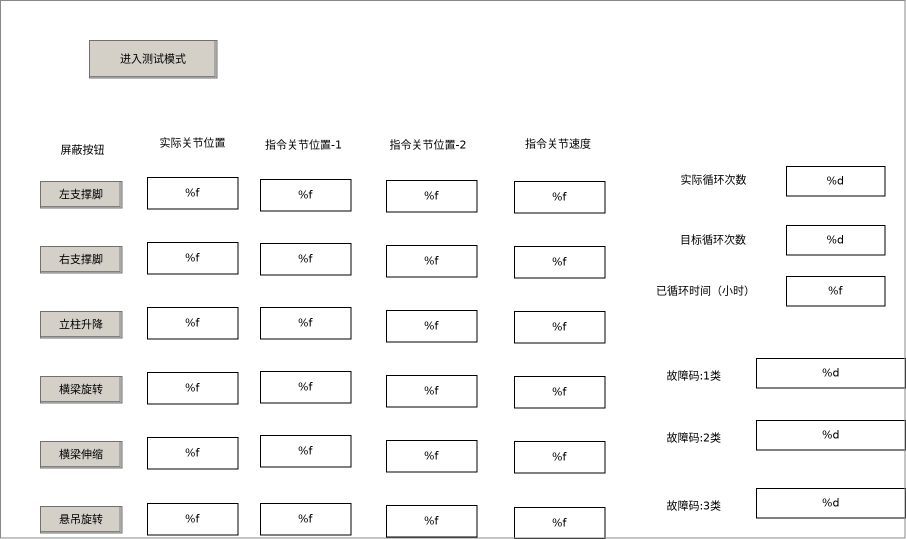
VISUALIZATION cartCycleTest  // 906x539
    Label (142,128 101x30), "实际关节位置"
    Rectangle (147,177 91x32), "%f", text variable: g_systemInfo.m_cartJntInfo[1].m_curJntPos
    Label (254,130 99x30), "指令关节位置-1"
    Button (89,40 128x38), "进入测试模式", colour toggle: g_cycleTest.m_carEnterCycleTest
        toggle g_cycleTest.m_carEnterCycleTest
    Rectangle (147,242 91x32), "%f", text variable: g_systemInfo.m_cartJntInfo[2].m_curJntPos
    Rectangle (260,179 91x32), "%f", text variable: g_cycleTest.m_targetJntPosCar[1][1]
        OnMouseClick: write the text variable via Default
    Rectangle (260,243 91x32), "%f", text variable: g_cycleTest.m_targetJntPosCar[1][2]
        OnMouseClick: write the text variable via Default
    Label (370,130 116x30), "指令关节位置-2"
    Rectangle (386,180 91x32), "%f", text variable: g_cycleTest.m_targetJntPosCar[2][1]
        OnMouseClick: write the text variable via Default
    Rectangle (386,245 91x32), "%f", text variable: g_cycleTest.m_targetJntPosCar[2][2]
        OnMouseClick: write the text variable via Default
    Rectangle (147,307 91x32), "%f", text variable: g_systemInfo.m_cartJntInfo[5].m_curJntPos
    Rectangle (147,372 91x32), "%f", text variable: g_systemInfo.m_cartJntInfo[6].m_curJntPos
    Rectangle (147,437 91x32), "%f", text variable: g_systemInfo.m_cartJntInfo[7].m_curJntPos
    Rectangle (147,503 91x32), "%f", text variable: g_systemInfo.m_cartJntInfo[8].m_curJntPos
    Rectangle (260,307 91x32), "%f", text variable: g_cycleTest.m_targetJntPosCar[1][5]
        OnMouseClick: write the text variable via Default
    Rectangle (260,371 91x32), "%f", text variable: g_cycleTest.m_targetJntPosCar[1][6]
        OnMouseClick: write the text variable via Default
    Rectangle (260,435 91x32), "%f", text variable: g_cycleTest.m_targetJntPosCar[1][7]
        OnMouseClick: write the text variable via Default
    Rectangle (260,503 91x32), "%f", text variable: g_cycleTest.m_targetJntPosCar[1][8]
        OnMouseClick: write the text variable via Default
    Rectangle (386,310 91x32), "%f", text variable: g_cycleTest.m_targetJntPosCar[2][5]
        OnMouseClick: write the text variable via Default
    Rectangle (386,375 91x32), "%f", text variable: g_cycleTest.m_targetJntPosCar[2][6]
        OnMouseClick: write the text variable via Default
    Rectangle (386,440 91x32), "%f", text variable: g_cycleTest.m_targetJntPosCar[2][7]
        OnMouseClick: write the text variable via Default
    Rectangle (386,505 91x32), "%f", text variable: g_cycleTest.m_targetJntPosCar[2][8]
        OnMouseClick: write the text variable via Default
    Label (507,130 102x28), "指令关节速度"
    Rectangle (514,181 91x32), "%f", text variable: g_cycleTest.m_targetJntVelCar[1]
        OnMouseClick: write the text variable via Default
    Rectangle (514,246 91x32), "%f", text variable: g_cycleTest.m_targetJntVelCar[2]
        OnMouseClick: write the text variable via Default
    Rectangle (514,311 91x32), "%f", text variable: g_cycleTest.m_targetJntVelCar[5]
        OnMouseClick: write the text variable via Default
    Rectangle (514,376 91x32), "%f", text variable: g_cycleTest.m_targetJntVelCar[6]
        OnMouseClick: write the text variable via Default
    Rectangle (514,441 91x32), "%f", text variable: g_cycleTest.m_targetJntVelCar[7]
        OnMouseClick: write the text variable via Default
    Rectangle (514,507 91x32), "%f", text variable: g_cycleTest.m_targetJntVelCar[8]
        OnMouseClick: write the text variable via Default
    Rectangle (786,225 99x30), "%d", text variable: g_cycleTest.m_targetCycleNumCar
        OnMouseClick: write g_cycleTest.m_targetCycleNumCar via Default
    Label (673,225 80x30), "目标循环次数"
    Rectangle (786,276 99x30), "%f", text variable: g_cycleTest.m_curCycleTimeCar
        OnMouseClick: write the text variable via Default
    Label (640,276 131x30), "已循环时间（小时）"
    Rectangle (756,358 150x30), "%d", text variable: GVL_interactUI.g_errIdType1
        OnMouseClick: write the text variable via Default
    Label (619,361 150x30), "故障码:1类"
    Rectangle (756,420 150x30), "%d", text variable: GVL_interactUI.g_errIdType2
        OnMouseClick: write the text variable via Default
    Label (619,423 150x30), "故障码:2类"
    Rectangle (756,488 150x30), "%d", text variable: GVL_interactUI.g_errIdType3
        OnMouseClick: write the text variable via Default
    Label (619,491 150x30), "故障码:3类"
    Rectangle (786,166 99x30), "%d", text variable: g_cycleTest.m_curCycleNumCar
        OnMouseClick: write CartControl.m_cartRobot.m_cartCycleTest.m_curCycleNum via Default
    Label (669,165 89x30), "实际循环次数"
    Button (40,181 82x27), "左支撑脚", colour toggle: g_cycleTest.m_disableCartJntMotion[1]
        toggle g_cycleTest.m_disableCartJntMotion[1]
    Button (40,246 82x27), "右支撑脚", colour toggle: g_cycleTest.m_disableCartJntMotion[2]
        toggle g_cycleTest.m_disableCartJntMotion[2]
    Button (40,311 82x27), "立柱升降", colour toggle: g_cycleTest.m_disableCartJntMotion[5]
        toggle g_cycleTest.m_disableCartJntMotion[5]
    Button (40,376 82x27), "横梁旋转", colour toggle: g_cycleTest.m_disableCartJntMotion[6]
        toggle g_cycleTest.m_disableCartJntMotion[6]
    Button (40,441 82x27), "横梁伸缩", colour toggle: g_cycleTest.m_disableCartJntMotion[7]
        toggle g_cycleTest.m_disableCartJntMotion[7]
    Button (40,506 82x27), "悬吊旋转", colour toggle: g_cycleTest.m_disableCartJntMotion[8]
        toggle g_cycleTest.m_disableCartJntMotion[8]
    Label (38,140 89x20), "屏蔽按钮"
END_VISUALIZATION

(* stored: Version 1.1.0.1, ProductVersion 3.1.4024.11
   Visu cartCycleTest: Id {023e9b0b-9b13-4b15-95cc-2be194297f02} *)
